// TIA Portal V20 export
DATA_BLOCK "DbMode"   // DB1
{ DB_Accessible_From_OPC_UA := 'FALSE' }
// stored: Access Published, DBAccessibleFromOPCUA false, MemoryReserve 100, Namespace LGeneral
   VAR
      operation { ExternalAccessible := 'False'; ExternalVisible := 'False'; ExternalWritable := 'False'} : Bool;
      operationON { ExternalAccessible := 'False'; ExternalVisible := 'False'; ExternalWritable := 'False'} : Bool;
      operationOFF { ExternalAccessible := 'False'; ExternalVisible := 'False'; ExternalWritable := 'False'} : Bool;
   END_VAR
BEGIN
END_DATA_BLOCK
